{attribute 'GeneratedUsingTerminal: EL4132--0000'}
{attribute addProperty BoxType "EL4132--0000"}
{attribute addProperty Id "EtcSlaveTerminalBaseChannel_1AT %Q*Channel_5F9B7EA62Channel_2AT %Q*Channel_5F9B7EA62WcStateAT %I*WcState_0B2B16F91InfoDataAT %I*InfoData_32EB74EA10"}
{attribute addProperty CRC "2346389980"}
{attribute addProperty Size "15"}
TYPE EL4132_8BDB11DC EXTENDS EtcSlaveTerminalBase :
STRUCT
	{attribute addProperty Name "Channel_1"}
	Channel_1 : Channel_5F9B7EA6;
	{attribute addProperty Name "Channel_2"}
	Channel_2 : Channel_5F9B7EA6;
	{attribute addProperty Name "WcState"}
	WcState : WcState_0B2B16F9;
	{attribute addProperty Name "InfoData"}
	InfoData : InfoData_32EB74EA;
END_STRUCT
END_TYPE

(* stored: Version 1.2.0.0, ProductVersion 3.1.4024.9
   DUT EL4132_8BDB11DC: Id {a38b363c-cf67-4273-8164-d33f930b1add} *)
